// Mitsubishi GX Works2 project: 2_3   PLC: FX1S

PROGRAM MAIN
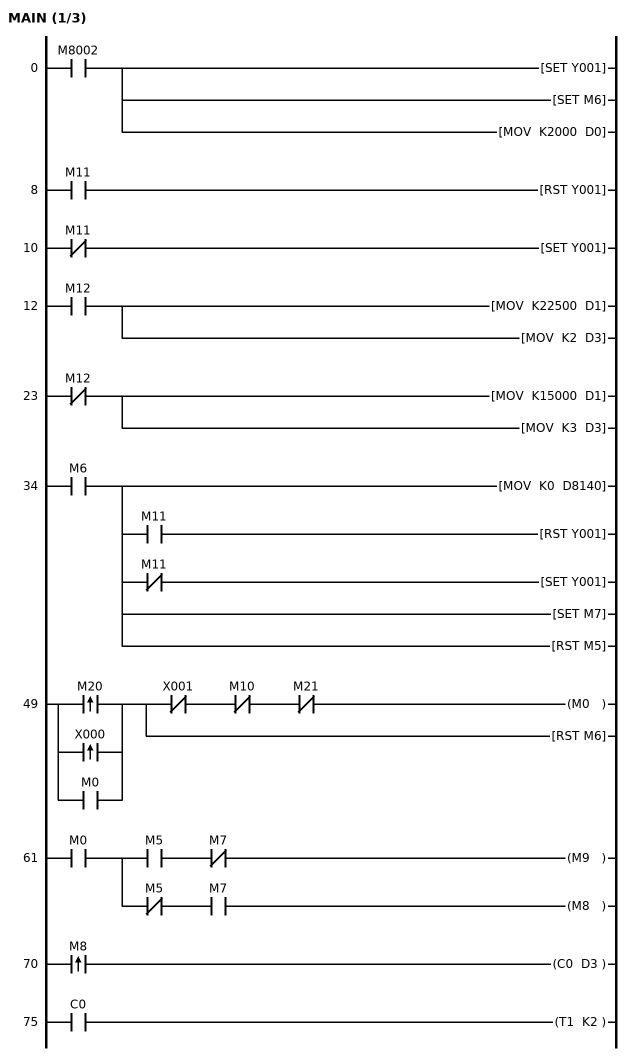
0     LD      M8002
      SET     Y001
      SET     M6
      MOV     K2000 D0
8     LD      M11
      RST     Y001
10    LDI     M11
      SET     Y001
12    LD      M12
      MOV     K22500 D1
      MOV     K2 D3
23    LDI     M12
      MOV     K15000 D1
      MOV     K3 D3
34    LD      M6
      MOV     K0 D8140
      MPS
      AND     M11
      RST     Y001
      MRD
      ANI     M11
      SET     Y001
      MPP
      SET     M7
      RST     M5
49    LDP     M20
      ORP     X000
      OR      M0
      MPS
      ANI     X001
      ANI     M10
      ANI     M21
      OUT     M0
      MPP
      RST     M6
61    LD      M0
      MPS
      AND     M5
      ANI     M7
      OUT     M9
      MPP
      ANI     M5
      AND     M7
      OUT     M8
70    LDP     M8
      OUT     C0 D3
75    LD      C0
      OUT     T1 K2
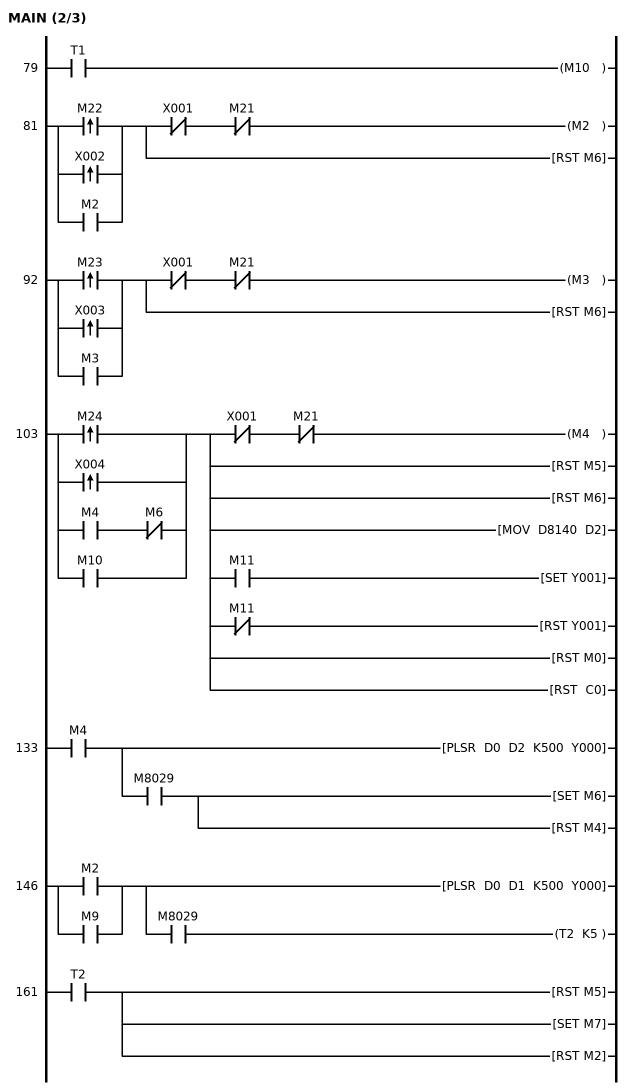
79    LD      T1
      OUT     M10
81    LDP     M22
      ORP     X002
      OR      M2
      MPS
      ANI     X001
      ANI     M21
      OUT     M2
      MPP
      RST     M6
92    LDP     M23
      ORP     X003
      OR      M3
      MPS
      ANI     X001
      ANI     M21
      OUT     M3
      MPP
      RST     M6
103   LDP     M24
      ORP     X004
      LD      M4
      ANI     M6
      ORB
      OR      M10
      MPS
      ANI     X001
      ANI     M21
      OUT     M4
      MPP
      RST     M5
      RST     M6
      MOV     D8140 D2
      MPS
      AND     M11
      SET     Y001
      MRD
      ANI     M11
      RST     Y001
      MPP
      RST     M0
      RST     C0
133   LD      M4
      PLSR    D0 D2 K500 Y000
      AND     M8029
      SET     M6
      RST     M4
146   LD      M2
      OR      M9
      PLSR    D0 D1 K500 Y000
      AND     M8029
      OUT     T2 K5
161   LD      T2
      RST     M5
      SET     M7
      RST     M2
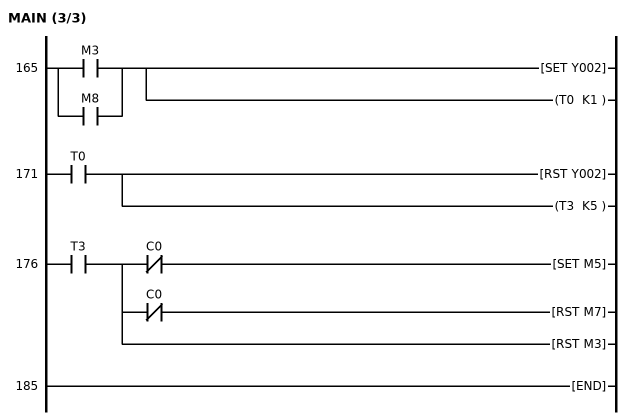
165   LD      M3
      OR      M8
      SET     Y002
      OUT     T0 K1
171   LD      T0
      RST     Y002
      OUT     T3 K5
176   LD      T3
      MPS
      ANI     C0
      SET     M5
      MRD
      ANI     C0
      RST     M7
      MPP
      RST     M3
185   END
END_PROGRAM
